Omron CX-Programmer project NewProject (CX-Programmer 9.75)

# PLC WATER_TANK_PROJECT: CJ2M CPU11

## Global symbols (name address type ; comment)
0.00 BOOL  ; AUTO/MANUAL
0.01 BOOL  ; START
0.02 BOOL  ; STOP
0.03 BOOL  ; LLS
0.04 BOOL  ; HLS
100.00 BOOL  ; L1
50.00 BOOL  ; M1
50.01 BOOL  ; M1

## Program NewProgram1 (cyclic task 0)

### Section Section1

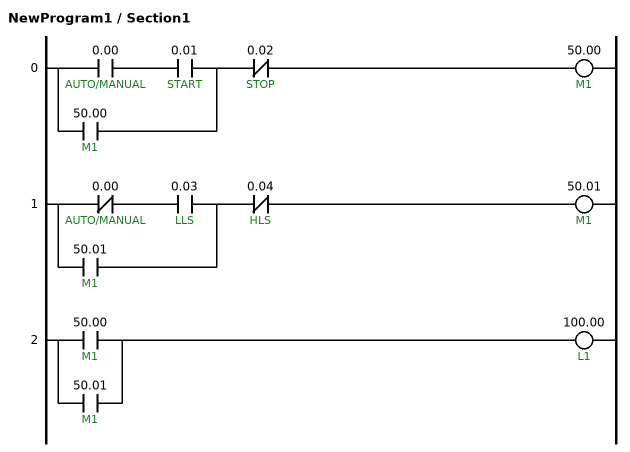
; rung 0
LD 0.00  ; AUTO/MANUAL
AND 0.01  ; START
OR 50.00  ; M1
ANDNOT 0.02  ; STOP
OUT 50.00  ; M1
; rung 1
LDNOT 0.00  ; AUTO/MANUAL
AND 0.03  ; LLS
OR 50.01  ; M1
ANDNOT 0.04  ; HLS
OUT 50.01  ; M1
; rung 2
LD 50.00  ; M1
OR 50.01  ; M1
OUT 100.00  ; L1

### Section END
; rung 0
END(001)